// TIA Portal V17 export
// export: Created 2025-03-07T09:16:42.8544205Z, ExportSetting WithDefaults, DisplayName Totally Integrated Automation Portal, DisplayVersion V17 Update 8, DisplayName TIA Portal Openness, DisplayVersion V17 Update 8, DisplayName TIA Portal Version Control Interface, DisplayVersion V17, DisplayName SINAMICS Startdrive Advanced, DisplayVersion V17 SP2, DisplayName SINAMICS Startdrive G110M, G120, G120C, G120D, G120P, G115D, DisplayVersion V17 SP2, DisplayName SINAMICS Startdrive G130, G150, S120, S150, SINAMICS MV, S210, DisplayVersion V17 SP2, DisplayName STEP 7 Professional, DisplayVersion V17 Update 8, DisplayName SINUMERIK ONE STEP 7 Toolbox, DisplayVersion V17 Update 12, DisplayName SINUMERIK 840D sl STEP 7 Toolbox, DisplayVersion V17 Update 12, DisplayName STEP 7 Safety, DisplayVersion V17 Update 6, DisplayName WinCC Advanced, DisplayVersion V17 Update 8
DATA_BLOCK "DB2441_MACHINE_STATUS"   // DB2441
{ S7_Optimized_Access := 'FALSE'; DB_Accessible_From_OPC_UA := 'FALSE' }
VERSION : 0.1
// stored: AutoNumber false, DBAccessibleFromOPCUA false, DBAccessibleFromWebserver true, IsOnlyStoredInLoadMemory false, IsWriteProtectedInAS false
   VAR RETAIN
      U01_IN_CLADDING : Bool;   // UNIT 01 STATION 3 CLADDING IN PROCESS
      U02_IN_CLADDING : Bool;   // UNIT 02 STATION 3 CLADDING IN PROCESS
      TIMER_U01_CLADDING : TOF_TIME;   // TIMER UNIT 01 STATION 3 CLADDING IN PROCESS OFF DELAY
      TIMER_U02_CLADDING : TOF_TIME;   // TIMER UNIT 02 STATION 3 CLADDING IN PROCESS OFF DELAY
   END_VAR
BEGIN
   TIMER_U01_CLADDING.PT := T#1s;
   TIMER_U02_CLADDING.PT := T#1s;
END_DATA_BLOCK
